PROGRAM MAIN
VAR
END_VAR

END_PROGRAM

(* stored: Version 1.1.0.1
   POU MAIN: Id {5d0e1a42-4235-491c-b56d-15ed7fcd0d91} *)
